// Mitsubishi GX Works2 project: conv   PLC: Q03UDV

PROGRAM MAIN
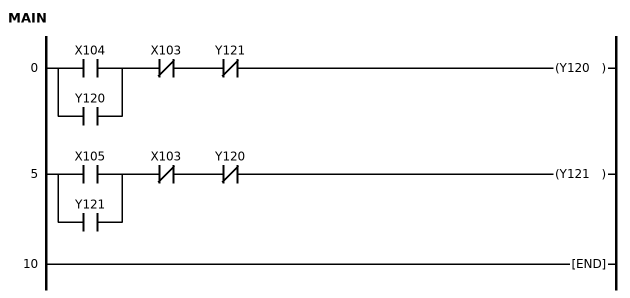
0     LD      X104
      OR      Y120
      ANI     X103
      ANI     Y121
      OUT     Y120
5     LD      X105
      OR      Y121
      ANI     X103
      ANI     Y120
      OUT     Y121
10    END
END_PROGRAM
